Fanuc KAREL source: kt00548.KL

-- PROVISIONAL review KL for V940-1; original PC SHA256 390ccd5b7871a9412723ae1b4af0c9f55d6219f1f3dd4774b688acb35cf6d492
-- Incomplete behavior may be omitted. Consult companion uncertainty JSON. Do not deploy.
PROGRAM KT00548
%NOLOCKGROUP
VAR
  OUT : BOOLEAN
-- UNRESOLVED_DECL P1 type=000199
-- UNRESOLVED_DECL P2 type=000199
BEGIN
  -- V9_ZERO_TABLE_METADATA_HINT layout=0001; no indexed target words; source/name/runtime held
  -- UNRESOLVED_PC offsets 5-38; opcodes 49,7E,49,7E,AC,23
  -- UNRESOLVED_PC offsets 43-47; opcodes 7F
END KT00548
